TYPE T_Char : STRING(1); END_TYPE

(* stored: Version 1.1.0.1, ProductVersion 3.1.4024.4
   DUT T_Char: Id {c7ed61be-fcbf-4958-8297-7ac57d7a6b68} *)
